PROGRAM PRG_Almacen
VAR
	iPosicion : INT;
	i: INT := 1;
	
	ALMACEN: INT;
	fTrigRRefSensorAlmacen	: F_TRIG;
	fTrigLift				: F_TRIG;
	fTrigMovingX			: F_TRIG;
	LECTURA: COLOR;
	DINT_TO_COLOR: DINT_TO_COLOR;
	bEstoyLleno: BOOL;
	tTimerRack : TON;

END_VAR

fTrigRRefSensorAlmacen(CLK:= GVL_Almacen.bRRflexSensorAlmacen);
fTrigLift(CLK:= GVL_Almacen.sStackCraneRack.MovingZ);
fTrigMovingX(CLK:= GVL_Almacen.sStackCraneRack.MovingX);
tTimerRack(IN:=GVL_Almacen.sStackCraneRack.MiddleLimit, PT:=T#1S);

CASE ALMACEN OF
	0:
	(* Colocamos el almacen en posición de espera *)
	
	GVL_Almacen.sStackCraneRack.TargetPosition := 55;
	GVL_Almacen.bLoadingConveyor := FALSE;
	
	IF NOT GVL_Almacen.sStackCraneRack.MovingX AND NOT GVL_Almacen.sStackCraneRack.MovingZ AND tTimerRack.Q THEN
		GVL_Almacen.sStackCraneRack.Right := TRUE;
		GVL_Almacen.sStackCraneRack.Lift  := FALSE;
	END_IF
	
	IF GVL_Almacen.sStackCraneRack.RightLimit THEN
		ALMACEN := 1;
	END_IF
	
	
	1:
	(* Esperamos a montar el palet en el almacén *)
	
	IF GVL_Almacen.iVisionSensorAlmacen > 0 THEN
		DINT_TO_COLOR(ENTRADA:= GVL_Almacen.iVisionSensorAlmacen, SALIDA=> LECTURA);
		GVL_Almacen.bLoadingConveyor := TRUE;
	END_IF

	IF fTrigRRefSensorAlmacen.Q THEN
		GVL_Almacen.bLoadingConveyor := FALSE;
		GVL_Almacen.sStackCraneRack.Lift:= TRUE;
	END_IF
	
	IF fTrigLift.Q THEN
		GVL_Almacen.sStackCraneRack.Right := FALSE;
	END_IF
	
	IF GVL_Almacen.sStackCraneRack.MiddleLimit THEN
		ALMACEN := 2;
	END_IF
	
	
	2:
	(* Una vez colocada la caja en posición, buscamos un sitio donde almacenar *)

	FOR i := 1 TO 54 BY 1 DO
		IF	GVL_Almacen.aAlmacen[i] = VACIO THEN
			iPosicion := i;
			GVL_Almacen.aAlmacen[i] := LECTURA;
			ALMACEN := 3;
			EXIT;
		ELSIF i = 54 THEN
			bEstoyLleno := TRUE;
			ALMACEN := 4;
		END_IF
	END_FOR
	
	
	3:
	(* Almacenamos en el sitio indicado *)
	
	GVL_Almacen.sStackCraneRack.TargetPosition := iPosicion;
	
	IF fTrigMovingX.Q THEN
		GVL_Almacen.sStackCraneRack.Left := TRUE;
	END_IF
	
	IF GVL_Almacen.sStackCraneRack.LeftLimit THEN
		GVL_Almacen.sStackCraneRack.Lift := FALSE;
		ALMACEN := 5;
	END_IF	
	
	
	5:
	(* Almacen lleno *)
	
	IF fTrigLift.Q THEN
		GVL_Almacen.sStackCraneRack.Left := FALSE;	
	END_IF
	
	IF GVL_Almacen.sStackCraneRack.MiddleLimit THEN
		ALMACEN := 0;
	END_IF
	
	
	4:
	(* Almacen lleno *)
	
	GVL_ProcesoPalet.sRollerConveyor.bRollerAlmacen2 := FALSE;
	GVL_ProcesoPalet.sRollerConveyor.bCurvedRollerAlmacen := FALSE;
	GVL_ProcesoPalet.sRollerConveyor.bRollerAlmacen1 := FALSE;
	
	IF NOT bEstoyLleno THEN
		ALMACEN := 0;
	END_IF
	
END_CASE

END_PROGRAM

(* stored: Version 1.1.0.1, ProductVersion 3.1.4024.12
   POU PRG_Almacen: Id {1101874a-6a42-4c7a-9ad2-e9048f62be9e}, SpecialFunc None *)
